// TwinCAT 3 PLC project ads_read_write_sample
// ProgramVersion: 3.1.4024.0
// libraries:
//   Tc2_Standard, * (Beckhoff Automation GmbH)
//   Tc2_System, * (Beckhoff Automation GmbH)
//   Tc3_Module, * (Beckhoff Automation GmbH)
// project tree:
//   DUTs/ ST_Sample.TcDUT
//   / PlcTask.TcTTO
//   POUs/ ADS_Write.TcPOU, ADS_Read.TcPOU, EIP_COM.TcPOU
// real-time tasks:
//   TASK PlcTask: cycle T#10ms, priority 20, ADS port 350
// I/O:
//   DEVICE Device 1 (TC3 EIP Adapter), AmsNetId 169.254.170.186.2.1
//     Box 1 (TC EtherNet/IP Slave)
// variable links:
//   ads_read_write_sample/ads_read_write_sample Instance <-> Device 1 (TC3 EIP Adapter)/Box 1 (TC EtherNet/IP Slave)
//     PlcTask Inputs/EIP_COM.eip_input <-> Assembly 1 (Input/Output)/Inputs/values
//     PlcTask Outputs/EIP_COM.eip_output <-> Assembly 1 (Input/Output)/Outputs/values

CONFIGURATION ads_read_write_sample
    RESOURCE PLC ON TwinCAT3
        TASK PlcTask(INTERVAL := T#10ms, PRIORITY := 20);
        PROGRAM ADS_Read WITH PlcTask : ADS_Read;
        PROGRAM ADS_Write WITH PlcTask : ADS_Write;
        PROGRAM EIP_COM WITH PlcTask : EIP_COM;
    END_RESOURCE
END_CONFIGURATION

// ---- DUTs/ST_Sample.TcDUT
TYPE ST_sample :
STRUCT
	title : STRING;
	id : UINT;
	datetime : DT;
END_STRUCT
END_TYPE

// ---- POUs/ADS_Read.TcPOU
PROGRAM ADS_Read
VAR
	fbReadReq  : ADSREADEX := ( NETID := '', PORT := 851, TMOUT := DEFAULT_ADS_TIMEOUT );
    bIncrement : BOOL;(* Rising edge at this variable starts command execution *)
    bDecrement : BOOL;(* Rising edge at this variable starts command execution *)
    bReset     : BOOL;(* Rising edge at this variable starts command execution *)
    bOther     : BOOL;(* Rising edge at this variable starts command execution *)
    
    nReadState     : BYTE;
    bBusy      : BOOL;
    bError     : BOOL;
    nErrID     : UDINT;
    cbRead     : UDINT;
    
    nCounter   : INT;(* Server data to be read *)
	stSample	: ST_Sample;
	bGetStructure: BOOL;
	
	


END_VAR

fbReadReq.NETID := '5.143.107.166.1.1'; // CX7000 target NetID

CASE nReadState OF
    0:
        IF bIncrement OR bDecrement OR bReset OR bOther OR bGetStructure THEN
            bBusy := TRUE;
            bError := FALSE;
            nErrID := 0;
            
            fbReadReq( READ := FALSE );

            IF bIncrement THEN(* Incement counter value *)
                bIncrement := FALSE;
                fbReadReq( IDXGRP := 16#8E000001, IDXOFFS := 0, LEN := SIZEOF(nCounter), DESTADDR := ADR(nCounter), READ := TRUE );
            ELSIF bDecrement THEN(* Decrement counter value *)
                bDecrement := FALSE;
                fbReadReq( IDXGRP := 16#8E000002, IDXOFFS := 0, LEN := SIZEOF(nCounter), DESTADDR := ADR(nCounter), READ := TRUE );
            ELSIF bReset THEN(* Reset counter value *)
                bReset := FALSE;
                fbReadReq( IDXGRP := 16#8E000003, IDXOFFS := 0, LEN := SIZEOF(nCounter), DESTADDR := ADR(nCounter), READ := TRUE );
			ELSIF bGetStructure THEN
				bGetStructure := FALSE;
				fbReadReq( IDXGRP := 16#8E000004, IDXOFFS := 0, LEN := SIZEOF(stSample), DESTADDR := ADR(stSample), READ := TRUE );
            ELSIF bOther THEN(* Call unsupported function *)
                bOther := FALSE;
                fbReadReq( IDXGRP := 16#8E000005, IDXOFFS := 0, LEN := SIZEOF(nCounter), DESTADDR := ADR(nCounter), READ := TRUE );
            END_IF
            
            nReadState := 1;
        END_IF
    1:
        fbReadReq( READ := FALSE, BUSY=>bBusy, ERR=>bError, ERRID=>nErrID, COUNT_R=>cbRead );
        IF NOT bBusy THEN
            IF NOT bError THEN
                nReadState := 0;(* Success *)
            ELSE
                nReadState := 100;(* Error *)
            END_IF
        END_IF
        
    100:(* TODO::Implement error handler *)
        nReadState := 0;
        
END_CASE

END_PROGRAM

// ---- POUs/ADS_Write.TcPOU
PROGRAM ADS_Write
VAR
	fbWriteReq   : ADSWRITE := ( NETID := '', PORT := 851, TMOUT := DEFAULT_ADS_TIMEOUT );
	bWrite       : BOOL;(* Rising edge at this variable starts command execution *)
	nWriteState  : BYTE;
	bBusy        : BOOL;
	bError       : BOOL;
	nErrID       : UDINT;
	arrInt       : ARRAY[0..9] OF INT;(* Server data to be written *)
	i            : INT;
END_VAR

fbWriteReq.NETID := '5.143.107.166.1.1'; // CX7000 target NetID

FOR i := 0 TO 9 DO
	arrInt[i] := i;
END_FOR

CASE nWriteState OF
	
   0:
      IF bWrite THEN
         bWrite := FALSE;
         
         bBusy := TRUE;
         bError := FALSE;
         nErrID := 0;
         
         fbWriteReq( WRITE := FALSE );
         fbWriteReq( IDXGRP := 16#80000005, IDXOFFS := 0, 
                  LEN := SIZEOF( arrInt ), SRCADDR := ADR( arrInt ), 
                  WRITE := TRUE );
         nWriteState := 1;            
      END_IF
      
   1:
      fbWriteReq( WRITE := FALSE, BUSY=>bBusy, ERR=>bError, ERRID=>nErrID );
      IF NOT bBusy THEN
         IF NOT bError THEN
            nWriteState := 0;(* Success *)
         ELSE
            nWriteState := 100;(* Error *)
         END_IF
      END_IF

   100:(* TODO::Implement error handler *)
      nWriteState := 0;
   
END_CASE

END_PROGRAM

// ---- POUs/EIP_COM.TcPOU
PROGRAM EIP_COM
VAR
	eip_input AT%I* : ARRAY [0..63] OF BYTE;
	eip_output AT%Q* : ARRAY [0..63] OF BYTE;

END_VAR

eip_output := eip_input;

END_PROGRAM
